{attribute 'OPC.UA.DA' := '1'}
FUNCTION_BLOCK FW212CAttenuationFilter EXTENDS AttenuationFilterBase
VAR_INPUT
END_VAR
VAR_OUTPUT
END_VAR
VAR
	{attribute 'OPC.UA.DA' := '0'}
	_config : FW212CAttenuationFilterConfig;
	{attribute 'OPC.UA.DA' := '0'}
	_coeAccess : CoeAccess;
	{attribute 'OPC.UA.DA' := '0'}
	_initConfigSerialCom : BOOL;	
	{attribute 'OPC.UA.DA' := '0'}
	_serialCom  : SerialCom(Prefix :='', Suffix := Const.CARRIAGE_RETURN);
	{attribute 'OPC.UA.DA' := '0'}
	_refSerialCom : REFERENCE TO SerialCom(Prefix :='', Suffix := Const.CARRIAGE_RETURN) := _serialCom;	 
	{attribute 'OPC.UA.DA' := '0'}
	_isReceived : BOOL;
	
	{attribute 'OPC.UA.DA' := '0'}
	_deliverMessages : INT;
	
	CheckConnectionMsg : STRING(255);
	PositionMsg : STRING(255);
	PositionCountMsg : STRING(255);
	IdMsg : STRING(255);
	CustomMsg : STRING(255);
	
	{region 'Commands'}	
		 
	{attribute 'OPC.UA.DA' := '0'}
	_moveAbsPosition	 : BOOL;
	{attribute 'OPC.UA.DA' := '0'}
	_jogBackwardPosition : BOOL;
	{attribute 'OPC.UA.DA' := '0'}
	_jogForwardPosition  : BOOL;
	{attribute 'OPC.UA.DA' := '0'}
	_customCmd : BOOL;
	{attribute 'OPC.UA.DA' := '0'}			  		   
	_raiseProperties : BOOL;
		 
	{attribute 'OPC.UA.DA' := '0'}
	_calibrateCmd : BOOL;
		 				  
	{endregion}
	
	{attribute 'OPC.UA.DA' := '0'}
	_initDevice : BOOL;	
	 
	{attribute 'OPC.UA.DA' := '0'}
	_pos : LREAL;
	{attribute 'OPC.UA.DA' := '0'}
	_cmd : STRING;	
	{attribute 'OPC.UA.DA' := '0'}
	_itemScheduler : INT;		
	{attribute 'OPC.UA.DA' := '0'}
	_pulseGenerator : TON;	
		
	{attribute 'OPC.UA.DA' := '0'}
	tmpMessage : STRING;	
	{attribute 'OPC.UA.DA' := '0'}
	message : STRING;
	{attribute 'OPC.UA.DA' := '0'}
	_length : INT;		 
	{attribute 'OPC.UA.DA' := '0'}
	_findSuffix : INT;
		
	{attribute 'OPC.UA.DA' := '0'}
	_calibrateStartAngle : LREAL;
	{attribute 'OPC.UA.DA' := '0'}
	_calibrateEndAngle : LREAL;
	{attribute 'OPC.UA.DA' := '0'}
	_angleSteps : LREAL;
	{attribute 'OPC.UA.DA' := '0'}
	_numberAverages : UINT;
	{attribute 'OPC.UA.DA' := '0'}
	_itemCalibrateScheduler : INT;
	{attribute 'OPC.UA.DA' := '0'}
	_itemRaisedProperties : INT;	
	
	{attribute 'OPC.UA.DA' := '0'}
	_itemPos : UINT;
	{attribute 'OPC.UA.DA' := '0'}
	_pulseCalibration : TON;	
	
	{region 'Calibrate'}
	
	{attribute 'OPC.UA.DA' := '0'}
	PowerMsg : STRING;
	{endregion}
			 	
	{attribute 'OPC.UA.DA' := '0'}
	_isOpen : BOOL;
	{attribute 'OPC.UA.DA' := '0'}
	_isWriteClose : BOOL;
	{attribute 'OPC.UA.DA' := '0'}
	ValuesCalibrate : ARRAY [0..1000] OF LREAL;
	{attribute 'OPC.UA.DA' := '0'}
	_counter : UINT;
	{attribute 'OPC.UA.DA' := '0'}
	PowerSum : LREAL;
	{attribute 'OPC.UA.DA' := '0'}
	PowerAverage : LREAL;
	
	{attribute 'OPC.UA.DA' := '0'}
	_pulseMoveGenerator : TON;
	{attribute 'OPC.UA.DA' := '0'}
	_itemMove : INT;
END_VAR


IF NOT InitConfigSerialCom THEN	
	ConfigureSerialCom();
ELSIF THIS^.Status = TExecutionState.Ready THEN	
	IF _refSerialCom.ErrorReceiveId = COMERROR_NOERROR THEN
		_refSerialCom(TxBuffer:= HardwareGlobalVariables.TxBufferAttenuation, 
			 	      RxBuffer:= HardwareGlobalVariables.RxBufferAttenuation);
	END_IF	
	
	// Init device
	InitDevice(); 				  
				  
	// Deliver messages
	IF _refSerialCom.IsReceived THEN
		CASE _deliverMessages OF			
			EFeedbackMsgAttenuationFW212C.CheckConnectionMsg :
				CheckConnectionMsg := _refSerialCom.LastReceivedString;	
			EFeedbackMsgAttenuationFW212C.PositionMsg :
				tmpMessage := DELETE(_refSerialCom.LastReceivedString, 6, 1);
				_length := LEN(tmpMessage);
				_findSuffix := FIND(tmpMessage, Const.CARRIAGE_RETURN);
				message := DELETE(tmpMessage, 4, _findSuffix);	
				
				PositionMsg := message;				
			EFeedbackMsgAttenuationFW212C.PositionCountMsg :
				PositionCountMsg := _refSerialCom.LastReceivedString;
			EFeedbackMsgAttenuationFW212C.IdMsg :
				IdMsg := _refSerialCom.LastReceivedString;
			EFeedbackMsgAttenuationFW212C.CustomMsg :
				CustomMsg := _refSerialCom.LastReceivedString;						
		END_CASE
		
		_deliverMessages := 0;
	END_IF						   	
					
	MoveAbsPosition(_moveAbsPosition, _pos);	
	JogBackwardPosition(_jogBackwardPosition);				
	JogForwardPosition(_jogForwardPosition);
	CustomCommand(_customCmd, _cmd);	
	RaisePropertiesChanged(_raiseProperties);

	IF (NOT _moveAbsPosition AND NOT _jogBackwardPosition AND NOT _jogForwardPosition AND NOT _customCmd
		AND NOT _raiseProperties AND _deliverMessages <> EFeedbackMsgAttenuationFW212C.PositionMsg) THEN
		MessageScheduler();
	END_IF	
END_IF

METHOD CheckConnection
VAR_INPUT
END_VAR
VAR
	cmd : STRING := '';
END_VAR
_deliverMessages := EFeedbackMsgAttenuationFW212C.CheckConnectionMsg;	
_serialCom.Send(cmd);
END_METHOD

METHOD ConfigureSerialCom
VAR_INPUT
END_VAR
VAR
END_VAR
IF _coeAccess.CoeOperation.Ready THEN
	_logger.Information(_message.Reset().Append('Start configuration com serial').ToString());
END_IF;	

_coeAccess.CoeOperation.Start();
_coeAccess(SerialCommunication := _config.SerialCommunication);
	
IF _coeAccess.CoeOperation.Done THEN
	_coeAccess.SetDone();	
 
	_Logger.Information(_message.Reset().
							Append('{').Append(TO_STRING(THIS^.Family)).Append('} : ').
							Append(' - Status : ').Append(TO_STRING(_coeAccess.Status)).ToString());	
	InitConfigSerialCom := TRUE;
END_IF
 
IF _coeAccess.CoeOperation.Error THEN	
	_coeAccess.SetError(0);
	
	_Logger.Error(_message.Reset().
							Append('{').Append(TO_STRING(THIS^.Family)).Append('} : ').
							Append(' - Status : ').Append(TO_STRING(_coeAccess.Status)).ToString());
	InitConfigSerialCom := TRUE;
END_IF

THIS^.Status := _coeAccess.Status;
State := _coeAccess.Status;
END_METHOD

{attribute 'TcRpcEnable' := '1'}
METHOD CustomCommand
VAR_INPUT
	Execute : BOOL;
	Cmd : STRING;
END_VAR
IF Execute THEN
	_logger.Information(_message.Reset().
								Append(_config.Name).
								Append(' - Custom : ').
								Append(Cmd).ToString());
	_deliverMessages := EFeedbackMsgAttenuationFW212C.CustomMsg;									
	_serialCom.Send(Cmd);
	
	_customCmd := FALSE;
END_IF
END_METHOD

METHOD FB_init : BOOL
VAR_INPUT
	bInitRetains : BOOL; // if TRUE, the retain variables are initialized (warm start / cold start)
	bInCopyCode : BOOL;  // if TRUE, the instance afterwards gets moved into the copy code (online change)
	Config : FW212CAttenuationFilterConfig;
END_VAR
VAR
END_VAR
IF Config.IsEnabled THEN
	_config := Config;
	
	SUPER^._attenuationFilterConfig.Name := Config.Name;
	SUPER^._attenuationFilterConfig.DeviceID := Config.DeviceID;
	SUPER^._attenuationFilterConfig.IsEnabled := Config.IsEnabled;
	SUPER^._attenuationFilterConfig.LogLevel := Config.LogLevel;
	
	SUPER^.Name := Config.Name;
	SUPER^.DeviceID := Config.DeviceID;	
	THIS^.Family := DeviceFamily.AttenuationFilter;
	
	_Logger.Information(_message.Reset().Append('Init ').
							Append('{').Append(TO_STRING(THIS^.Family)).Append('} - ').
							Append('{').Append(TO_STRING(Config.Name)).Append('}').ToString());																													
END_IF
END_METHOD

(** Returns the model number and firmware version **)
METHOD GetIdentifier
VAR_INPUT
END_VAR
VAR
	cmd : STRING := '*idn?';
END_VAR
_deliverMessages := EFeedbackMsgAttenuationFW212C.IdMsg;
_serialCom.Send(cmd);
END_METHOD

(** Position Query **)
METHOD PROTECTED GetPosition
VAR_INPUT
END_VAR
VAR
	cmd : STRING := 'pos?';
END_VAR
_deliverMessages := EFeedbackMsgAttenuationFW212C.PositionMsg;
_serialCom.Send(cmd);
END_METHOD

(** Returns the wheel type **)
METHOD GetPositionCount
VAR_INPUT
END_VAR
VAR
	cmd : STRING := 'pcount?';
END_VAR
_deliverMessages := EFeedbackMsgAttenuationFW212C.PositionCountMsg;
_serialCom.Send(cmd);
END_METHOD

PROPERTY InitConfigSerialCom : BOOL
GET
InitConfigSerialCom := _initConfigSerialCom;
END_GET
SET
_initConfigSerialCom := InitConfigSerialCom;
END_SET
END_PROPERTY

METHOD InitDevice 
VAR_INPUT
END_VAR
VAR
END_VAR
IF NOT _initDevice THEN	
	_logger.Information(_message.Reset().
								Append(_config.Name).
								Append(' - Init device').ToString());
										
	// TODO : define max count 
	_itemScheduler := 10;
	
	_initDevice := TRUE;	
END_IF
END_METHOD

{attribute 'TcRpcEnable' := '1'}
(** Decrements the filter position by 1 **)
METHOD PROTECTED JogBackwardPosition
VAR_INPUT
	Execute : BOOL;
END_VAR
VAR
	jogBackwardPos : BYTE := 68;
	posArray       : ARRAY[1..3] OF BYTE := [27, 91, jogBackwardPos];	
END_VAR
IF Execute THEN
	_jogBackwardPosition := TRUE;

	IF _pulseMoveGenerator.Q THEN	
		CASE _itemMove OF							
			0:	_logger.Information(_message.Reset().
											Append(_config.Name).
											Append(' - Jog backward position').ToString());
					
				_serialCom.Send3B(posArray);
				
				_itemMove := 1;
				
			1:  GetPosition();
				_itemMove := 10;	
								
			10:  _jogBackwardPosition := FALSE;
				_itemMove := 0;			
		END_CASE			
	ELSE
		_pulseMoveGenerator(IN := TRUE, PT := T#200MS);	
	END_IF	
END_IF
END_METHOD

{attribute 'TcRpcEnable' := '1'}
(** Increments the filter position by 1 **)
METHOD PROTECTED JogForwardPosition
VAR_INPUT
	Execute : BOOL;
END_VAR
VAR
	jogForwardPos : BYTE := 67;
	posArray      : ARRAY[1..3] OF BYTE := [27, 91, jogForwardPos];
END_VAR
IF Execute THEN
	_jogForwardPosition := TRUE;

	IF _pulseMoveGenerator.Q THEN	
		CASE _itemMove OF							
			0:	_logger.Information(_message.Reset().
											Append(_config.Name).
											Append(' - Jog forward position').ToString());
					
				_serialCom.Send3B(posArray);
				
				_itemMove := 1;
				
			1:  GetPosition();
				_itemMove := 10;	
								
			10:  _jogForwardPosition := FALSE;
				_itemMove := 0;			
		END_CASE			
	ELSE
		_pulseMoveGenerator(IN := TRUE, PT := T#200MS);	
	END_IF	
END_IF
END_METHOD

METHOD MessageScheduler
VAR_INPUT
END_VAR
IF _pulseGenerator.Q THEN
	_pulseGenerator(IN := FALSE, PT := T#10MS);
		
	CASE _itemScheduler OF	
		10:	GetPosition();
			_itemScheduler := 0;
			
		1:  GetPositionCount();
			_itemScheduler := 2;
			
		2:  CheckConnection();
			_itemScheduler := 3;

		3:  GetIdentifier();
			_itemScheduler := 0;								
	END_CASE
ELSE
	_pulseGenerator(IN := TRUE, PT := T#100MS);	
END_IF
END_METHOD

{attribute 'TcRpcEnable' := '1'}
(** Absulute moves the wheel to filter position n **)
METHOD PROTECTED MoveAbsPosition 
VAR_INPUT
	Execute : BOOL;
	Position : LREAL;
END_VAR
VAR
	cmd : STRING := 'pos=';
	cmdConcat : STRING(255);
END_VAR
IF Execute THEN
	_moveAbsPosition := TRUE;

	IF _pulseMoveGenerator.Q THEN	
		CASE _itemMove OF							
			0:	_logger.Information(_message.Reset().
											Append(_config.Name).
											Append(' - Move absolute position : ').Append(TO_STRING(Position)).ToString());
					
				cmdConcat := CONCAT(cmd, TO_STRING(LREAL_TO_INT(Position)));
				_serialCom.Send(cmdConcat);
				
				_itemMove := 1;
				
			1:  GetPosition();
				_itemMove := 10;	
								
			10:  _moveAbsPosition := FALSE;
				_itemMove := 0;			
		END_CASE			
	ELSE
		_pulseMoveGenerator(IN := TRUE, PT := T#100MS);	
	END_IF	
END_IF
END_METHOD

{attribute 'TcRpcEnable' := '1'}
METHOD RaisePropertiesChanged
VAR_INPUT
	Execute : BOOL;
END_VAR
IF Execute THEN
	IF THIS^.Status <> TExecutionState.Ready THEN	
		_raiseProperties := FALSE;
		RETURN;
	END_IF	

	_raiseProperties := TRUE;
	
	IF _pulseGenerator.Q THEN
		_pulseGenerator(IN := FALSE, PT := T#10MS);	

		CASE _itemRaisedProperties OF
			0:	PositionMsg := ' ';
				
				_itemRaisedProperties := 10;
			
			10:  GetPosition();
				_itemRaisedProperties := 11;
							
			11:  _logger.Information(_message.Reset().
								Append(_config.Name).
								Append(' - Attenuation RaisePropertiesChanged').ToString());
				_raiseProperties := FALSE;				
				_itemRaisedProperties := 0;
			
		END_CASE
	ELSE
		_pulseGenerator(IN := TRUE, PT := T#100MS);	
	END_IF
END_IF
END_METHOD

END_FUNCTION_BLOCK

(* stored: Version 1.1.0.1, ProductVersion 3.1.4024.12
   POU FW212CAttenuationFilter: Id {400e0f4b-36e5-48c0-befe-a5516db9517d}, SpecialFunc None
   Folder Commands: Id {80efaf67-af5b-4b7c-bfbf-4581898e7be6}
   Method CheckConnection: Id {edfe6120-1a82-43da-a9d0-4f0250f661d3}
   Method ConfigureSerialCom: Id {d5934859-2097-4d5b-bc4c-1798adc04d2b}
   Method CustomCommand: Id {cb5a68f9-861d-41bc-b5c0-d84f275daf85}
   Method FB_init: Id {40470048-f926-4d48-8362-4c2b0f10d282}
   Method GetIdentifier: Id {b87a6ffc-50eb-4f8a-855a-9202528c91f5}
   Method GetPosition: Id {4388dade-acb0-4b55-b092-f53a71006226}
   Method GetPositionCount: Id {4250de32-6de9-4a4e-bbe5-7c24ee9d7ad3}
   Property InitConfigSerialCom: Id {74d81c74-6061-424f-946d-bdf55a29a503}
   Get Get: Id {06235796-f672-471f-97c4-9248ef8ffa15}
   Set Set: Id {2cb60bc0-b0f2-4d30-ac09-24b44cd69008}
   Method InitDevice: Id {be3876a0-d8b0-4848-8fbd-755108321599}
   Method JogBackwardPosition: Id {7420c2a6-b345-4d8a-90dc-f186735d5a93}
   Method JogForwardPosition: Id {62f276c8-040c-4d10-9c78-d2be385ec6cd}
   Method MessageScheduler: Id {147ac8b0-fdeb-4a50-a723-9e19f3a97bb8}
   Method MoveAbsPosition: Id {1687eab1-1c65-466a-9b30-40f99e03772f}
   Method RaisePropertiesChanged: Id {263c3c10-74e0-4b74-9091-37c6168cc450} *)
